TYPE ST_ProtectionSystems_set :
STRUCT
	//Fire Detection System
	FireDetection						: ST_Firedetection_set;
	
	//InsulationMonitor
	Insulation							: ST_InsulationMonitor_set;
	
	//OCP
	OvercurrentProtection				: ST_OvercurrentProtection_set;
END_STRUCT
END_TYPE

(* stored: Version 1.1.0.1, ProductVersion 3.1.4026.18
   DUT ST_ProtectionSystems_set: Id {b97d13dd-fe93-424a-9c1a-8b8a4082bd10} *)
